Fanuc KAREL source: IO0215.KL

-- PROVISIONAL review KL for V770-1; original PC SHA256 106b2bc69aebc76cf1acfdb17bb40c916eb8a5437e00a32bc9c43b8b4fae574a
-- Incomplete behavior may be omitted. Consult companion uncertainty JSON. Do not deploy.
PROGRAM IO0215
%NOLOCKGROUP
-- UNRESOLVED_LOCAL_POOL 5 cells at code offset 13; source declarations unknown
-- DIRECT_LOCAL_WORD_ACCESS alone does not prove INTEGER, REAL, or BOOLEAN
BEGIN
  -- UNRESOLVED_PC offsets 0-18; opcodes 2B,2C,7B
  -- UNRESOLVED_PC offsets 23-30; opcodes 9D,23
  -- UNRESOLVED_PC offsets 35-49; opcodes 2E,22,9D,33,35
  -- UNRESOLVED_PC offsets 54-61; opcodes 9D,23
  -- UNRESOLVED_PC offsets 66-77; opcodes 2E,23
  -- UNRESOLVED_PC offsets 82-107; opcodes 22,21,33,9D,33,36,4A
  -- UNRESOLVED_PC offsets 112-116; opcodes 7F
  -- UNRESOLVED_PC offsets 121-125; opcodes 27,AA
  -- UNRESOLVED_PC offsets 130-134; opcodes 7F
END IO0215
